// TIA Portal V16 export
// export: Created 2025-08-30T12:59:10.9026933Z, ExportSetting WithDefaults, DisplayName Totally Integrated Automation Portal, DisplayVersion V16, DisplayName TIA Portal Version Control Interface, DisplayVersion V16, DisplayName TIA Portal Openness, DisplayVersion V16, DisplayName STEP 7 Professional, DisplayVersion V16, DisplayName STEP 7 Safety, DisplayVersion V16, DisplayName WinCC Advanced, DisplayVersion V16
FUNCTION "Servo_DriveManager" : Void   // FC17, FBD
TITLE = Drive Manager Closed Loop
VERSION : 0.1
// Drive Manager for Closed Loop with Encoder
// stored: AutoNumber true, IsIECCheckEnabled false, UDAEnableTagReadback false
   VAR_INPUT
      "[NAME] Axis Name" : String;
      "[INPUT] ReferenceSwitch_Input" : Bool;
      "[INPUT] Drive Ready" : Bool;
      "[INPUT] E-STOP Check" : Bool;
      "[COMMAND] Start_Reference Run" : Bool;
      "[COMMAND] Take_over_Pos" : Bool;
      "[COMMAND] Go to Position" : Bool;
      "[COMMAND] Axis Manual Forward" : Bool;
      "[COMMAND] Axis Manual Reverse" : Bool;
      "[COMMAND] Axis Speed" : Int;
      "[COMMAND] Axis Fast Stop" : Bool;
      "[COMMAND] Go To Rest" : Bool;
      "[COMMAND] Axis Brake" : Bool;
      "[VALUE] Reference Position" : Int;
      "[VALUE] Set Position" : Real;
      "[VALUE] Rest Position" : Real;
      "[VALUE] Accelerating" : Real;
      "[VALUE] Deaccelerating" : Real;
      "[VALUE] Position Tolerance" : Real;
      "[COMMUNICATION] MasterWord" : String;
      "[COMMUNICATION] Callback" : String;
   END_VAR
   VAR_OUTPUT
      "[OUTPUT] Drive FWD Command" : Bool;
      "[OUTPUT] Drive REV Command" : Bool;
      "[OUTPUT] Drive Speed 2 (50%)" : Bool;
      "[OUTPUT] Drive Speed 3 (75%)" : Bool;
      "[OUTPUT] Drive Fast Stop Command" : Bool;
      "[MESSAGE] Axis Busy" : Bool;
      "[MESSAGE] Error Executing" : Bool;
      "[MESSAGE] Axis On Position" : Bool;
      "[MESSAGE] Axis On Rest" : Bool;
      "[MESSAGE] Drive State" : String;
      "[MESSAGE] Axis Slips" : String;
   END_VAR
   VAR_TEMP
      UnscPos : Int;
      ScPos : Real;
      ActEncPos : Real;
      SetRefRun : Bool;
      SetRefRun_Q : Bool;
      MoveToRest : Bool;
      MoveToRest_Q : Bool;
      Automatic_Positive : Bool;
      Manual_Positive : Bool;
      Automatic_Negative : Bool;
      Manual_Negative : Bool;
      HS_Positive : Bool;
      MasterWordHex : Int;
      Speed50 : Bool;
      Speed75 : Bool;
      Min_Position : Real;
      Max_Position : Real;
      Axis_On_Position : Bool;
      Direction_Forward : Bool;
      Direction_Backward : Bool;
      Drive_Auto_Fwd : Bool;
      InternalFastStop : Bool;
      RefRunSetSignal : Bool;
      GoToRest2 : Bool;
      "[COMMAND] Go to Position_Rest" : Bool;
      RestPos_SpareMove : Real;
   END_VAR
   VAR_TEMP   // added for the SCL form of the ladder/FBD networks
      _w1 : Bool;
   END_VAR
BEGIN

REGION Network 1: Reference Run
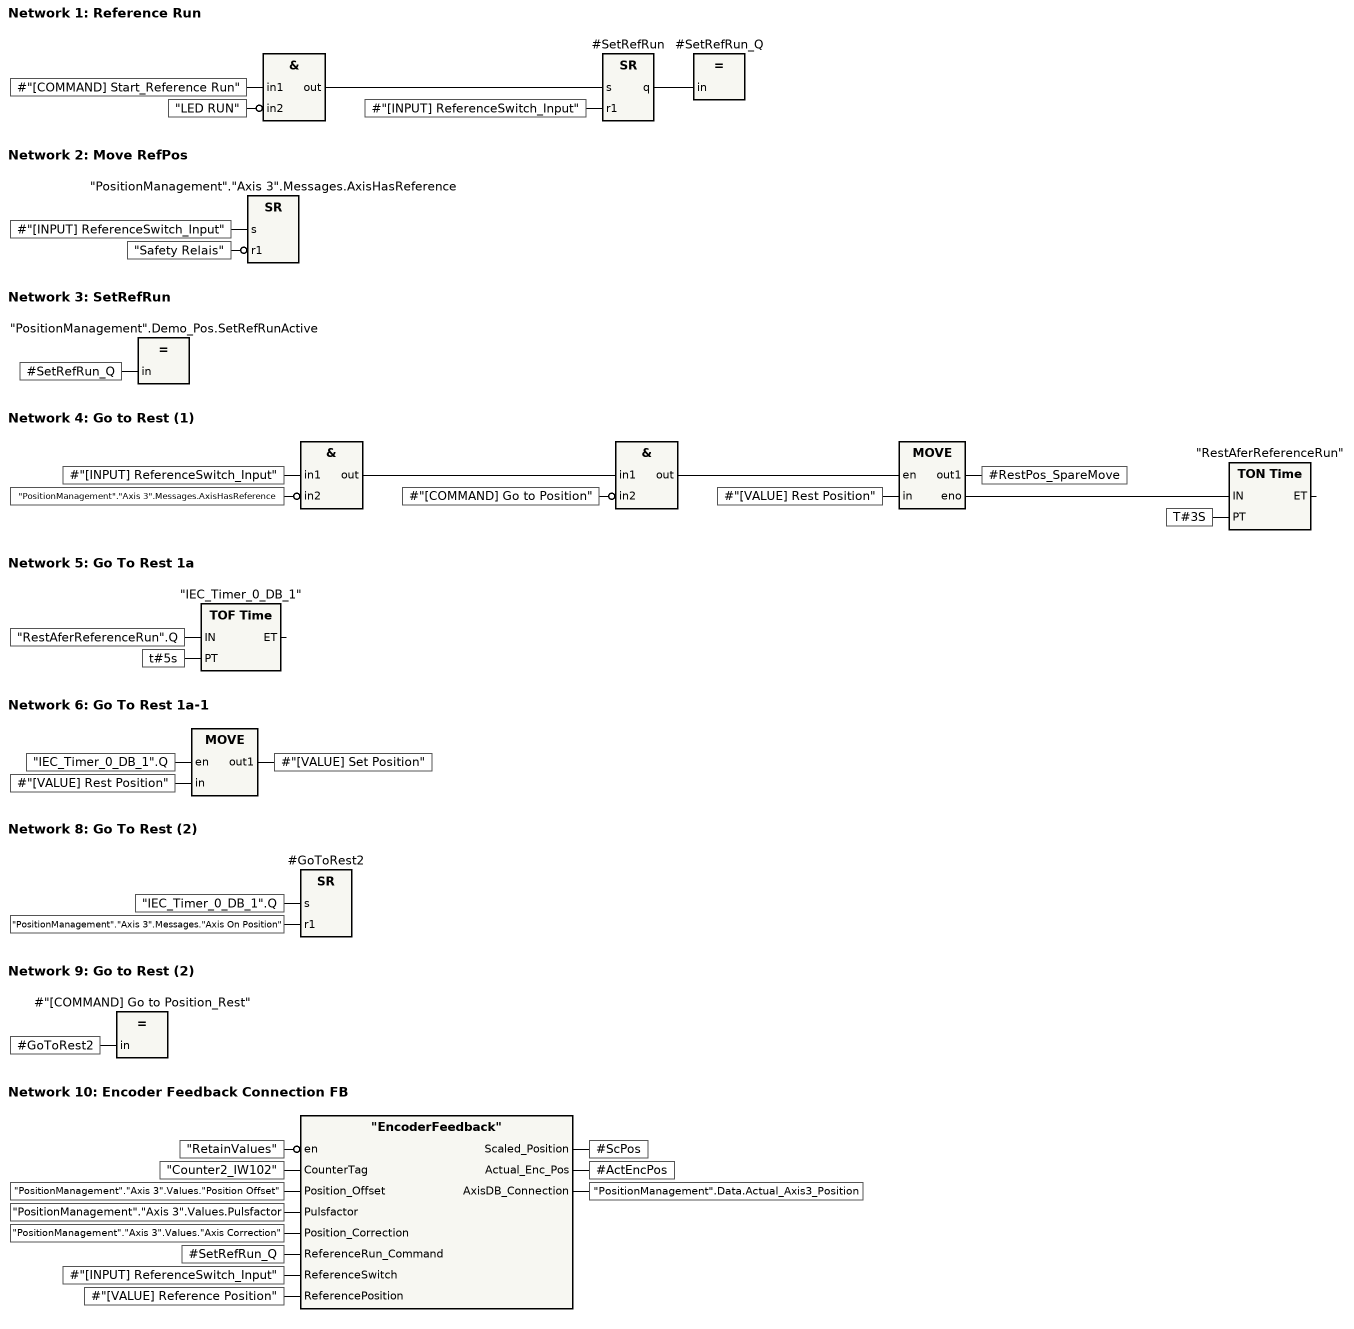
   IF #"[COMMAND] Start_Reference Run" AND NOT "LED RUN" THEN
       #SetRefRun := TRUE;   // SR flip-flop
   END_IF;
   IF #"[INPUT] ReferenceSwitch_Input" THEN #SetRefRun := FALSE; END_IF;
   #SetRefRun_Q := #SetRefRun;
END_REGION

REGION Network 2: Move RefPos
   IF #"[INPUT] ReferenceSwitch_Input" THEN
       "PositionManagement"."Axis 3".Messages.AxisHasReference := TRUE;   // SR flip-flop
   END_IF;
   IF NOT "Safety Relais" THEN "PositionManagement"."Axis 3".Messages.AxisHasReference := FALSE; END_IF;
END_REGION

REGION Network 3: SetRefRun
   "PositionManagement".Demo_Pos.SetRefRunActive := #SetRefRun_Q;
END_REGION

REGION Network 4: Go to Rest (1)
   // ENO of a box is taken as its EN; it also drops when the box reports an error
   #_w1 := #"[INPUT] ReferenceSwitch_Input" AND NOT "PositionManagement"."Axis 3".Messages.AxisHasReference AND NOT #"[COMMAND] Go to Position";
   IF #_w1 THEN #RestPos_SpareMove := #"[VALUE] Rest Position"; END_IF;
   "RestAferReferenceRun".TON(IN := #_w1, PT := T#3S);
END_REGION

REGION Network 5: Go To Rest 1a
   "IEC_Timer_0_DB_1".TOF(IN := "RestAferReferenceRun".Q, PT := t#5s);
END_REGION

REGION Network 6: Go To Rest 1a-1
   IF "IEC_Timer_0_DB_1".Q THEN #"[VALUE] Set Position" := #"[VALUE] Rest Position"; END_IF;
END_REGION

REGION Network 7: Go To Rest 1b
END_REGION

REGION Network 8: Go To Rest (2)
   IF "IEC_Timer_0_DB_1".Q THEN
       #GoToRest2 := TRUE;   // SR flip-flop
   END_IF;
   IF "PositionManagement"."Axis 3".Messages."Axis On Position" THEN #GoToRest2 := FALSE; END_IF;
END_REGION

REGION Network 9: Go to Rest (2)
   #"[COMMAND] Go to Position_Rest" := #GoToRest2;
END_REGION

REGION Network 10: Encoder Feedback Connection FB
   // Getting the feedback from the encoder device
   IF NOT "RetainValues" THEN
       "EncoderFeedback"(CounterTag := "Counter2_IW102",
                         Position_Offset := "PositionManagement"."Axis 3".Values."Position Offset",
                         Pulsfactor := "PositionManagement"."Axis 3".Values.Pulsfactor,
                         Position_Correction := "PositionManagement"."Axis 3".Values."Axis Correction",
                         ReferenceRun_Command := #SetRefRun_Q,
                         ReferenceSwitch := #"[INPUT] ReferenceSwitch_Input",
                         ReferencePosition := #"[VALUE] Reference Position",
                         Scaled_Position => #ScPos,
                         Actual_Enc_Pos => #ActEncPos,
                         AxisDB_Connection => "PositionManagement".Data.Actual_Axis3_Position);
   END_IF;
END_REGION

REGION Network 11: Calculate Position Tolerance 1
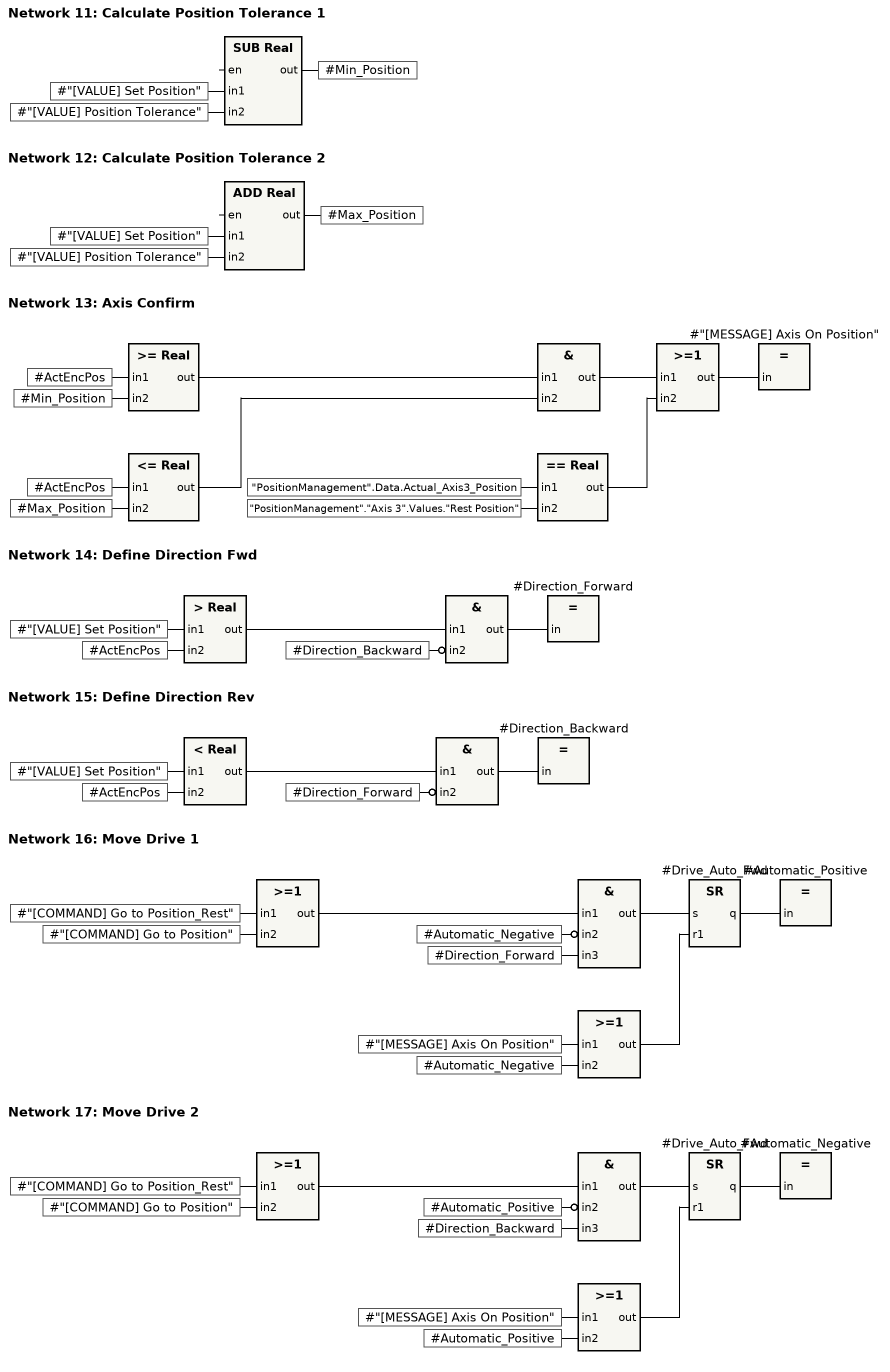
   #Min_Position := #"[VALUE] Set Position" - #"[VALUE] Position Tolerance";
END_REGION

REGION Network 12: Calculate Position Tolerance 2
   #Max_Position := #"[VALUE] Set Position" + #"[VALUE] Position Tolerance";
END_REGION

REGION Network 13: Axis Confirm
   #"[MESSAGE] Axis On Position" := ((#ActEncPos >= #Min_Position) AND (#ActEncPos <= #Max_Position)) OR ("PositionManagement".Data.Actual_Axis3_Position = "PositionManagement"."Axis 3".Values."Rest Position");
END_REGION

REGION Network 14: Define Direction Fwd
   #Direction_Forward := (#"[VALUE] Set Position" > #ActEncPos) AND NOT #Direction_Backward;
END_REGION

REGION Network 15: Define Direction Rev
   #Direction_Backward := (#"[VALUE] Set Position" < #ActEncPos) AND NOT #Direction_Forward;
END_REGION

REGION Network 16: Move Drive 1
   IF (#"[COMMAND] Go to Position_Rest" OR #"[COMMAND] Go to Position") AND NOT #Automatic_Negative AND #Direction_Forward THEN
       #Drive_Auto_Fwd := TRUE;   // SR flip-flop
   END_IF;
   IF #"[MESSAGE] Axis On Position" OR #Automatic_Negative THEN #Drive_Auto_Fwd := FALSE; END_IF;
   #Automatic_Positive := #Drive_Auto_Fwd;
END_REGION

REGION Network 17: Move Drive 2
   IF (#"[COMMAND] Go to Position_Rest" OR #"[COMMAND] Go to Position") AND NOT #Automatic_Positive AND #Direction_Backward THEN
       #Drive_Auto_Fwd := TRUE;   // SR flip-flop
   END_IF;
   IF #"[MESSAGE] Axis On Position" OR #Automatic_Positive THEN #Drive_Auto_Fwd := FALSE; END_IF;
   #Automatic_Negative := #Drive_Auto_Fwd;
END_REGION

REGION Network 18: Manual Displacement Positive
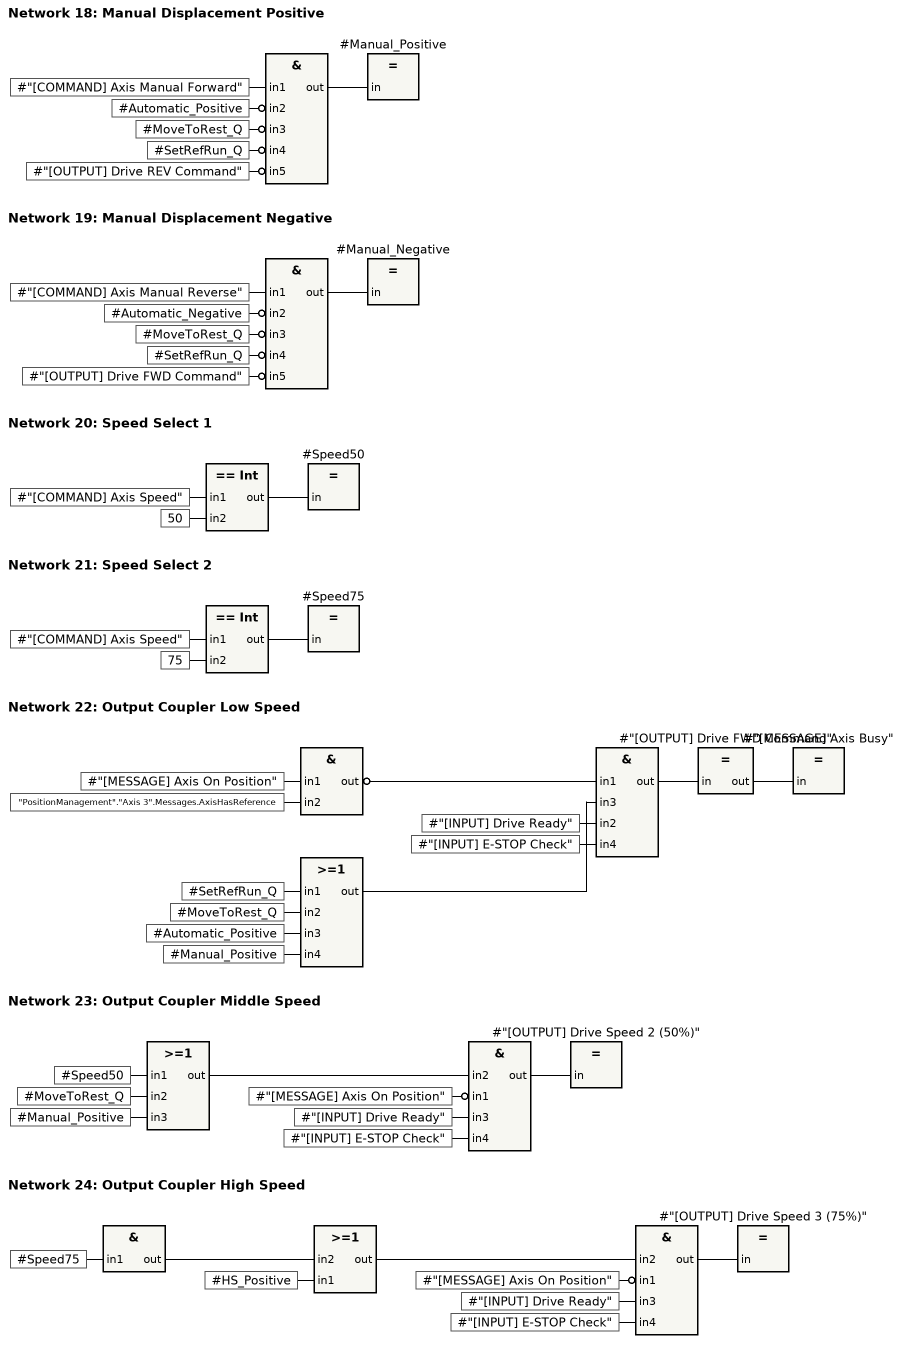
   #Manual_Positive := #"[COMMAND] Axis Manual Forward" AND NOT #Automatic_Positive AND NOT #MoveToRest_Q AND NOT #SetRefRun_Q AND NOT #"[OUTPUT] Drive REV Command";
END_REGION

REGION Network 19: Manual Displacement Negative
   #Manual_Negative := #"[COMMAND] Axis Manual Reverse" AND NOT #Automatic_Negative AND NOT #MoveToRest_Q AND NOT #SetRefRun_Q AND NOT #"[OUTPUT] Drive FWD Command";
END_REGION

REGION Network 20: Speed Select 1
   #Speed50 := #"[COMMAND] Axis Speed" = 50;
END_REGION

REGION Network 21: Speed Select 2
   #Speed75 := #"[COMMAND] Axis Speed" = 75;
END_REGION

REGION Network 22: Output Coupler Low Speed
   #_w1 := NOT (#"[MESSAGE] Axis On Position" AND "PositionManagement"."Axis 3".Messages.AxisHasReference) AND (#SetRefRun_Q OR #MoveToRest_Q OR #Automatic_Positive OR #Manual_Positive) AND #"[INPUT] Drive Ready" AND #"[INPUT] E-STOP Check";
   #"[OUTPUT] Drive FWD Command" := #_w1;
   #"[MESSAGE] Axis Busy" := #_w1;
END_REGION

REGION Network 23: Output Coupler Middle Speed
   #"[OUTPUT] Drive Speed 2 (50%)" := (#Speed50 OR #MoveToRest_Q OR #Manual_Positive) AND NOT #"[MESSAGE] Axis On Position" AND #"[INPUT] Drive Ready" AND #"[INPUT] E-STOP Check";
END_REGION

REGION Network 24: Output Coupler High Speed
   #"[OUTPUT] Drive Speed 3 (75%)" := (#Speed75 OR #HS_Positive) AND NOT #"[MESSAGE] Axis On Position" AND #"[INPUT] Drive Ready" AND #"[INPUT] E-STOP Check";
END_REGION

REGION Network 25: Output Coupler Reverse
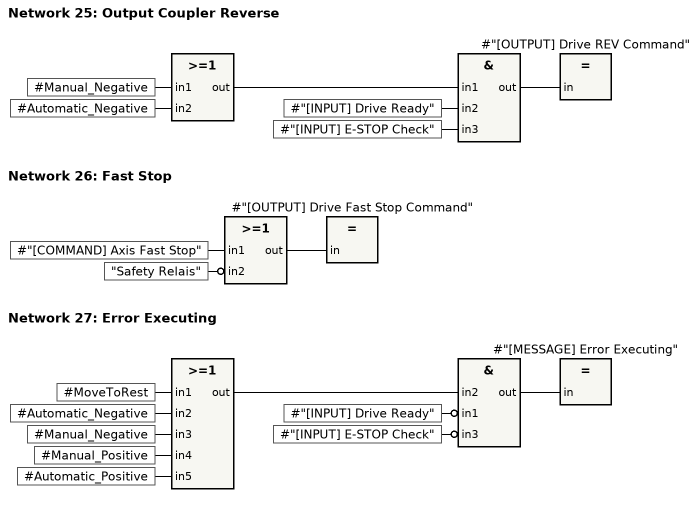
   #"[OUTPUT] Drive REV Command" := (#Manual_Negative OR #Automatic_Negative) AND #"[INPUT] Drive Ready" AND #"[INPUT] E-STOP Check";
END_REGION

REGION Network 26: Fast Stop
   #"[OUTPUT] Drive Fast Stop Command" := #"[COMMAND] Axis Fast Stop" OR NOT "Safety Relais";
END_REGION

REGION Network 27: Error Executing
   #"[MESSAGE] Error Executing" := (#MoveToRest OR #Automatic_Negative OR #Manual_Negative OR #Manual_Positive OR #Automatic_Positive) AND NOT #"[INPUT] Drive Ready" AND NOT #"[INPUT] E-STOP Check";
END_REGION
END_FUNCTION
